FUNCTION_BLOCK FB_DisplacementSensor

VAR_OUTPUT
	nDistance : INT;
	bInValueRange : BOOL;
END_VAR
VAR
	aInputBytes AT %I* : ARRAY[1..2] OF BYTE;
	nWord1 : WORD;
	nWord2 : WORD;
	nWord3 : WORD;
                                                                                                                                                                                                                                                                                                                                                                                                                                                                                                                                                                                                                                                                                                                                                                                                                                                                                                                                                                                                                                                                                                                                                                                                                                                                                                         I* : ARRAY 
END_VAR

nWord1 := TO_WORD(aInputBytes[1]);

//1111_1111
//0000_0000_1111_1111


nWord2 := aInputBytes[2];
//1111_1111
//0000_0000_1111_1111

nWord1 := SHL(nWord1, 8);
// 1111_1111_0000_0000
nWord3 := nWord1 OR nWord2;
//1111_1111_1111_1111
nWord3 := SHR(nWord3,4);

nDistance := TO_INT(nWord3); 

bInValueRange := aInputBytes[2].0;

END_FUNCTION_BLOCK

(* stored: Version 1.1.0.1, ProductVersion 3.1.4024.12
   POU FB_DisplacementSensor: Id {de668adf-6580-4528-8136-4c20d1b579d8}, SpecialFunc None *)
